FUNCTION_BLOCK FB_AirCylinder
VAR
    bEnable : BOOL;
END_VAR

END_FUNCTION_BLOCK

(* stored: POU FB_AirCylinder: Id {00000000-0000-0000-0000-000000000002} *)
